// TIA Portal project "FactoryIO_Template_S7-1200_V16_V16" (V16)
// Vorlageprojekt für das Buch mit Zielsystem S7-1200

(* hardware
DEVICE "S7-1200-Station_1"  S7-1200 Station
   slot 0: "Baugruppenträger_0"  Rack  V1.0
   slot 1: "PLC_1"  CPU 1211C DC/DC/DC  6ES7 211-1AE40-0XB0  V4.1
*)

// ===== PLC "PLC_1"  CPU 1211C DC/DC/DC =====

VAR_GLOBAL   // PLC tag table "Standard-Variablentabelle"
   "Tag_4" AT %I10.0 : Bool;
   "Tag_5" AT %Q10.0 : Bool;
   "Tag_6" AT %I10.1 : Bool;
   "loop marker" AT %M0.0 : Bool;
   "stop-cond" AT %M0.1 : Bool;
   "stop-cond-pulse" AT %M0.2 : Bool;
   "Tag_1" AT %M2.0 : Bool;
   "Tag_2" AT %M2.1 : Bool;
   "cancel-grap" AT %M0.3 : Bool;
   "return-X" AT %M0.4 : Bool;
   "reset-c" AT %M0.5 : Bool;
   "Tag_7" AT %M2.2 : Bool;
   "Tag_8" AT %M1.0 : Bool;
   "Tag_9" AT %M1.1 : Bool;
   "grab-control" AT %M0.6 : Bool;
   "Tag_3" AT %M2.3 : Bool;
   "Tag_10" AT %M2.4 : Bool;
   "Tag_11" AT %M1.2 : Bool;
   "shift palett" AT %M0.7 : Bool;
   "Tag_12" AT %M2.5 : Bool;
   "palett-c-reset" AT %M1.3 : Bool;
   "Tag_13" AT %M2.6 : Bool;
END_VAR

VAR_GLOBAL   // PLC tag table "Tag table from XML_1"
   "Start Button" AT %I0.0 : Bool;
   "Stop Button" AT %I0.1 : Bool;
   "Emergency Stop" AT %I0.2 : Bool;
   "Diffuse Sensor 1" AT %I0.3 : Bool;
   "Diffuse Sensor 2" AT %I0.4 : Bool;
   "Diffuse Sensor 3" AT %I0.5 : Bool;
   "Moving (Z) Detected" AT %I0.6 : Bool;
   "Moving (X) Detected" AT %I0.7 : Bool;
   "Detected" AT %I1.0 : Bool;
   "Belt Conveyor 1 (6m)" AT %Q0.0 : Bool;
   "Belt Conveyor 2 (6m)" AT %Q0.1 : Bool;
   "Belt Conveyor (4m)" AT %Q0.2 : Bool;
   "Roller Conveyor 1 (6m)" AT %Q0.3 : Bool;
   "Roller Conveyor 2 (6m)" AT %Q0.4 : Bool;
   "Roller Conveyor (4m)" AT %Q0.5 : Bool;
   "Moving (Z)" AT %Q0.6 : Bool;
   "Moving (X)" AT %Q0.7 : Bool;
   "Grab" AT %Q1.0 : Bool;
   "Start Button  (Light)" AT %Q1.1 : Bool;
   "Stop Button  (Light)" AT %Q1.2 : Bool;
END_VAR

// folder: System blocks/Program resources

DATA_BLOCK "palett-c"   // DB1
{ S7_Optimized_Access := 'TRUE' }
AUTHOR : Simatic
FAMILY : IEC
NAME : CNTR
VERSION : 1.0
// stored: InstanceOfName IEC_COUNTER
"IEC_COUNTER"
BEGIN
END_DATA_BLOCK

DATA_BLOCK "sequence-counter"   // DB2
{ S7_Optimized_Access := 'TRUE' }
AUTHOR : Simatic
FAMILY : IEC
NAME : CNTR
VERSION : 1.0
// stored: InstanceOfName IEC_COUNTER
"IEC_COUNTER"
BEGIN
END_DATA_BLOCK

DATA_BLOCK "palett-shift"   // DB3
{ S7_Optimized_Access := 'TRUE' }
AUTHOR : Simatic
FAMILY : IEC
NAME : IEC_TMR
VERSION : 1.0
// stored: InstanceOfName IEC_TIMER
"IEC_TIMER"
BEGIN
END_DATA_BLOCK

DATA_BLOCK "TT"   // DB4
{ S7_Optimized_Access := 'TRUE' }
AUTHOR : Simatic
FAMILY : IEC
NAME : IEC_TMR
VERSION : 1.0
// stored: InstanceOfName IEC_TIMER
"IEC_TIMER"
BEGIN
END_DATA_BLOCK

// folder: (top level)

FUNCTION "MHJ-PLC-Lab-Function-S71200" : Void   // FC9000, SCL
{ S7_Optimized_Access := 'TRUE' }
VERSION : 0.1
   VAR_TEMP
      rdTimeReturn : Int;
      outputTime : DTL;
      SyncVal : Byte;
      forVal : Int;
      forVal_2 : Int;
      Value : Byte;
   END_VAR
   VAR CONSTANT
      CompVal : Byte := 16#34;
      Value_01 : Byte := 16#11;
      Value_01_DW : DWord := 16#A165_D992;
      Value_02_DW : DWord := 16#58BE_4401;
   END_VAR
BEGIN

   #Value:=PEEK(area := 16#82,
        dbNumber := 0,
        byteOffset := 511);
   #Value := #Value + 1;

   POKE(area := 16#82,
        dbNumber := 0,
        byteOffset := 511,
        value := #Value);

   POKE(area:=16#81,
        dbNumber:=0,
        byteOffset:=1016,
        value:=#Value_01_DW);
   POKE(area := 16#81,
        dbNumber := 0,
        byteOffset := 1020,
        value := #Value_02_DW);

   POKE(area := 16#81,
        dbNumber := 0,
        byteOffset := 511,
        value := B#16#00);

   FOR #forVal := 0 TO 120 DO
       FOR #forVal_2:=0 TO 10 DO
           #rdTimeReturn:=RD_SYS_T(#outputTime);
           #rdTimeReturn := WR_SYS_T(#outputTime);
           #rdTimeReturn := RD_SYS_T(#outputTime);
           #rdTimeReturn := WR_SYS_T(#outputTime);
       END_FOR;
       #SyncVal:= PEEK(area := 16#81,
                      dbNumber := 0,
                      byteOffset := 511);
       IF #SyncVal = #CompVal THEN
          GOTO M_1;
       END_IF;
   END_FOR;
   RETURN;

   M_1:
   POKE(area := 16#81,
        dbNumber := 0,
        byteOffset := 511,
        value := B#16#0);
END_FUNCTION

ORGANIZATION_BLOCK "Main"   // OB1, LAD, ProgramCycle
TITLE = "Main Program Sweep (Cycle)"
{ S7_Optimized_Access := 'TRUE' }
VERSION : 0.1
   VAR_INPUT
      Initial_Call : Bool;   // Initial call of this OB
      Remanence : Bool;   // =True, if remanent data are available
   END_VAR
   VAR_TEMP   // added for the SCL form of the ladder/FBD networks
      _w1 : Bool;
      _w2 : Bool;
   END_VAR
BEGIN

REGION Network 1: Konnektierungsbaustein für PLC-Lab
   // Im Netzwerk 1 wird der Konnektierungsbaustein für PLC-Lab aufgerufen.
   // Dieser Aufruf darf nicht entfernt werden!
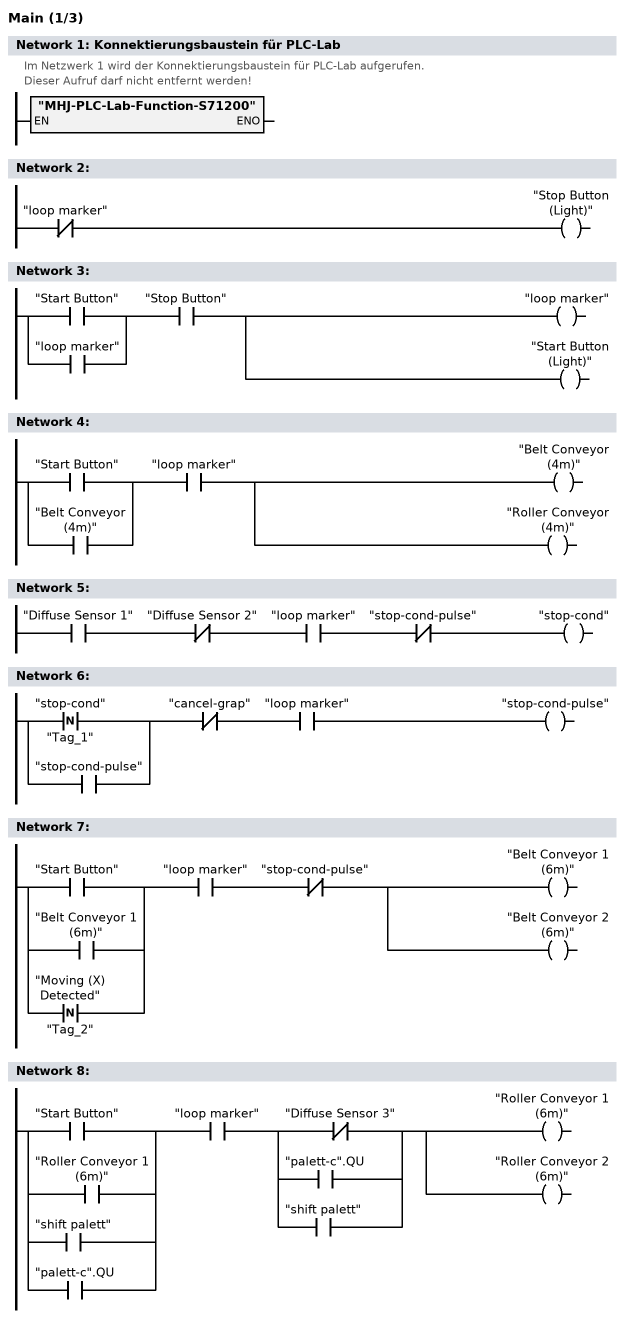
   RUNG wire#powerrail
      "MHJ-PLC-Lab-Function-S71200"()
   END_RUNG
   // the same network as SCL:
   "MHJ-PLC-Lab-Function-S71200"();
END_REGION

REGION Network 2
   RUNG wire#powerrail
      I_Contact( "loop marker" )
      Coil( "Stop Button  (Light)" )
   END_RUNG
   // the same network as SCL:
   "Stop Button  (Light)" := NOT "loop marker";
END_REGION

REGION Network 3
   RUNG wire#powerrail
      Contact( "Start Button" )
      wire#w1
      Contact( "Stop Button" )
      wire#w2
      Coil( "loop marker" )
   END_RUNG
   RUNG wire#powerrail
      Contact( "loop marker" )
   END_RUNG wire#w1
   RUNG wire#w2
      Coil( "Start Button  (Light)" )
   END_RUNG
   // the same network as SCL:
   "loop marker" := ("Start Button" OR "loop marker") AND "Stop Button";
   "Start Button  (Light)" := "loop marker";
END_REGION

REGION Network 4
   RUNG wire#powerrail
      Contact( "Start Button" )
      wire#w1
      Contact( "loop marker" )
      wire#w2
      Coil( "Belt Conveyor (4m)" )
   END_RUNG
   RUNG wire#powerrail
      Contact( "Belt Conveyor (4m)" )
   END_RUNG wire#w1
   RUNG wire#w2
      Coil( "Roller Conveyor (4m)" )
   END_RUNG
   // the same network as SCL:
   "Belt Conveyor (4m)" := ("Start Button" OR "Belt Conveyor (4m)") AND "loop marker";
   "Roller Conveyor (4m)" := "Belt Conveyor (4m)";
END_REGION

REGION Network 5
   RUNG wire#powerrail
      Contact( "Diffuse Sensor 1" )
      I_Contact( "Diffuse Sensor 2" )
      Contact( "loop marker" )
      I_Contact( "stop-cond-pulse" )
      Coil( "stop-cond" )
   END_RUNG
   // the same network as SCL:
   "stop-cond" := "Diffuse Sensor 1" AND NOT "Diffuse Sensor 2" AND "loop marker" AND NOT "stop-cond-pulse";
END_REGION

REGION Network 6
   RUNG wire#powerrail
      N_Contact(operand := "stop-cond", bit := "Tag_1")
      wire#w1
      I_Contact( "cancel-grap" )
      Contact( "loop marker" )
      Coil( "stop-cond-pulse" )
   END_RUNG
   RUNG wire#powerrail
      Contact( "stop-cond-pulse" )
   END_RUNG wire#w1
   // the same network as SCL:
   #_w1 := NOT "stop-cond" AND "Tag_1";   // falling edge of "stop-cond"
   "Tag_1" := "stop-cond";
   "stop-cond-pulse" := (#_w1 OR "stop-cond-pulse") AND NOT "cancel-grap" AND "loop marker";
END_REGION

REGION Network 7
   RUNG wire#powerrail
      Contact( "Start Button" )
      wire#w1
      Contact( "loop marker" )
      I_Contact( "stop-cond-pulse" )
      wire#w2
      Coil( "Belt Conveyor 1 (6m)" )
   END_RUNG
   RUNG wire#powerrail
      Contact( "Belt Conveyor 1 (6m)" )
   END_RUNG wire#w1
   RUNG wire#powerrail
      N_Contact(operand := "Moving (X) Detected", bit := "Tag_2")
   END_RUNG wire#w1
   RUNG wire#w2
      Coil( "Belt Conveyor 2 (6m)" )
   END_RUNG
   // the same network as SCL:
   #_w1 := NOT "Moving (X) Detected" AND "Tag_2";   // falling edge of "Moving (X) Detected"
   "Tag_2" := "Moving (X) Detected";
   "Belt Conveyor 1 (6m)" := ("Start Button" OR "Belt Conveyor 1 (6m)" OR #_w1) AND "loop marker" AND NOT "stop-cond-pulse";
   "Belt Conveyor 2 (6m)" := "Belt Conveyor 1 (6m)";
END_REGION

REGION Network 8
   RUNG wire#powerrail
      Contact( "Start Button" )
      wire#w1
      Contact( "loop marker" )
      wire#w2
      I_Contact( "Diffuse Sensor 3" )
      wire#w3
      Coil( "Roller Conveyor 1 (6m)" )
   END_RUNG
   RUNG wire#powerrail
      Contact( "Roller Conveyor 1 (6m)" )
   END_RUNG wire#w1
   RUNG wire#powerrail
      Contact( "shift palett" )
   END_RUNG wire#w1
   RUNG wire#powerrail
      Contact( "palett-c".QU )
   END_RUNG wire#w1
   RUNG wire#w2
      Contact( "palett-c".QU )
   END_RUNG wire#w3
   RUNG wire#w2
      Contact( "shift palett" )
   END_RUNG wire#w3
   RUNG wire#w3
      Coil( "Roller Conveyor 2 (6m)" )
   END_RUNG
   // the same network as SCL:
   "Roller Conveyor 1 (6m)" := ("Start Button" OR "Roller Conveyor 1 (6m)" OR "shift palett" OR "palett-c".QU) AND "loop marker" AND (NOT "Diffuse Sensor 3" OR "palett-c".QU OR "shift palett");
   "Roller Conveyor 2 (6m)" := "Roller Conveyor 1 (6m)";
END_REGION

REGION Network 9
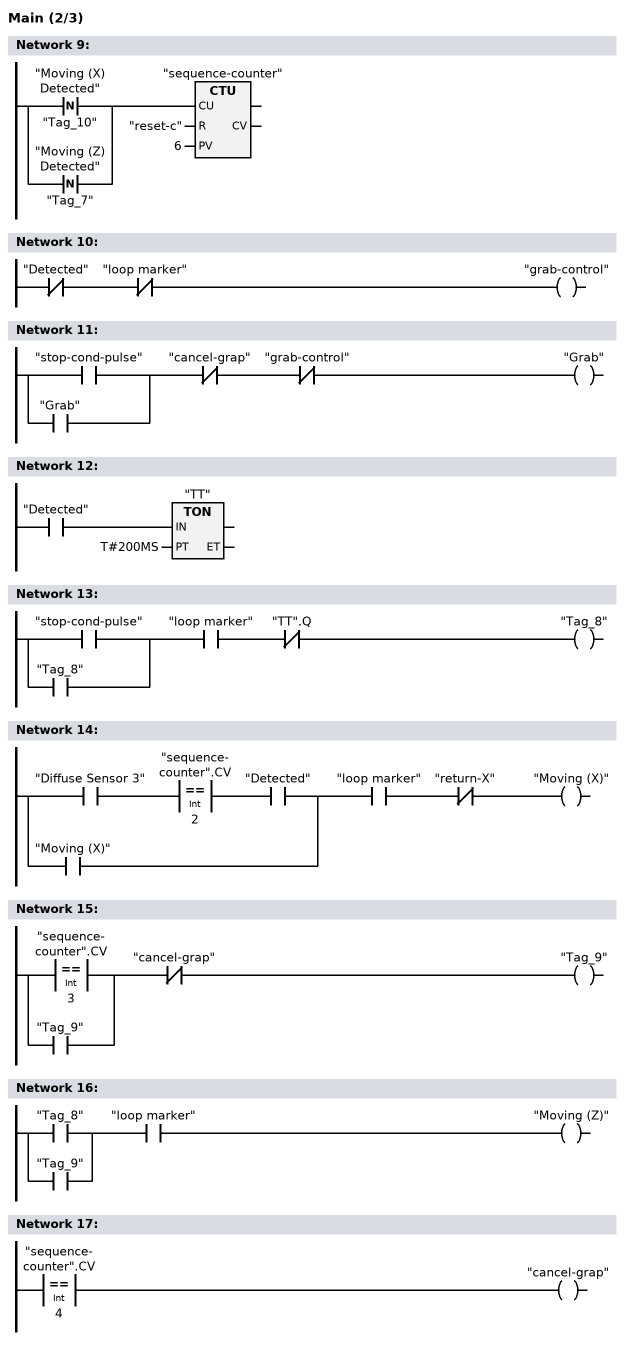
   #_w1 := NOT "Moving (X) Detected" AND "Tag_10";   // falling edge of "Moving (X) Detected"
   "Tag_10" := "Moving (X) Detected";
   #_w2 := NOT "Moving (Z) Detected" AND "Tag_7";   // falling edge of "Moving (Z) Detected"
   "Tag_7" := "Moving (Z) Detected";
   "sequence-counter".CTU(CU := #_w1 OR #_w2, R := "reset-c", PV := 6);
END_REGION

REGION Network 10
   RUNG wire#powerrail
      I_Contact( "Detected" )
      I_Contact( "loop marker" )
      Coil( "grab-control" )
   END_RUNG
   // the same network as SCL:
   "grab-control" := NOT "Detected" AND NOT "loop marker";
END_REGION

REGION Network 11
   RUNG wire#powerrail
      Contact( "stop-cond-pulse" )
      wire#w1
      I_Contact( "cancel-grap" )
      I_Contact( "grab-control" )
      Coil( "Grab" )
   END_RUNG
   RUNG wire#powerrail
      Contact( "Grab" )
   END_RUNG wire#w1
   // the same network as SCL:
   "Grab" := ("stop-cond-pulse" OR "Grab") AND NOT "cancel-grap" AND NOT "grab-control";
END_REGION

REGION Network 12
   "TT".TON(IN := "Detected", PT := T#200MS);
END_REGION

REGION Network 13
   RUNG wire#powerrail
      Contact( "stop-cond-pulse" )
      wire#w1
      Contact( "loop marker" )
      I_Contact( "TT".Q )
      Coil( "Tag_8" )
   END_RUNG
   RUNG wire#powerrail
      Contact( "Tag_8" )
   END_RUNG wire#w1
   // the same network as SCL:
   "Tag_8" := ("stop-cond-pulse" OR "Tag_8") AND "loop marker" AND NOT "TT".Q;
END_REGION

REGION Network 14
   RUNG wire#powerrail
      Contact( "Diffuse Sensor 3" )
      { S7_Templates := "SrcType := Int" } EQ_Contact(in1 := "sequence-counter".CV, in2 := 2)
      Contact( "Detected" )
      wire#w1
      Contact( "loop marker" )
      I_Contact( "return-X" )
      Coil( "Moving (X)" )
   END_RUNG
   RUNG wire#powerrail
      Contact( "Moving (X)" )
   END_RUNG wire#w1
   // the same network as SCL:
   "Moving (X)" := (("Diffuse Sensor 3" AND ("sequence-counter".CV = 2) AND "Detected") OR "Moving (X)") AND "loop marker" AND NOT "return-X";
END_REGION

REGION Network 15
   RUNG wire#powerrail
      { S7_Templates := "SrcType := Int" } EQ_Contact(in1 := "sequence-counter".CV, in2 := 3)
      wire#w1
      I_Contact( "cancel-grap" )
      Coil( "Tag_9" )
   END_RUNG
   RUNG wire#powerrail
      Contact( "Tag_9" )
   END_RUNG wire#w1
   // the same network as SCL:
   "Tag_9" := (("sequence-counter".CV = 3) OR "Tag_9") AND NOT "cancel-grap";
END_REGION

REGION Network 16
   RUNG wire#powerrail
      Contact( "Tag_8" )
      wire#w1
      Contact( "loop marker" )
      Coil( "Moving (Z)" )
   END_RUNG
   RUNG wire#powerrail
      Contact( "Tag_9" )
   END_RUNG wire#w1
   // the same network as SCL:
   "Moving (Z)" := ("Tag_8" OR "Tag_9") AND "loop marker";
END_REGION

REGION Network 17
   RUNG wire#powerrail
      { S7_Templates := "SrcType := Int" } EQ_Contact(in1 := "sequence-counter".CV, in2 := 4)
      Coil( "cancel-grap" )
   END_RUNG
   // the same network as SCL:
   "cancel-grap" := "sequence-counter".CV = 4;
END_REGION

REGION Network 18
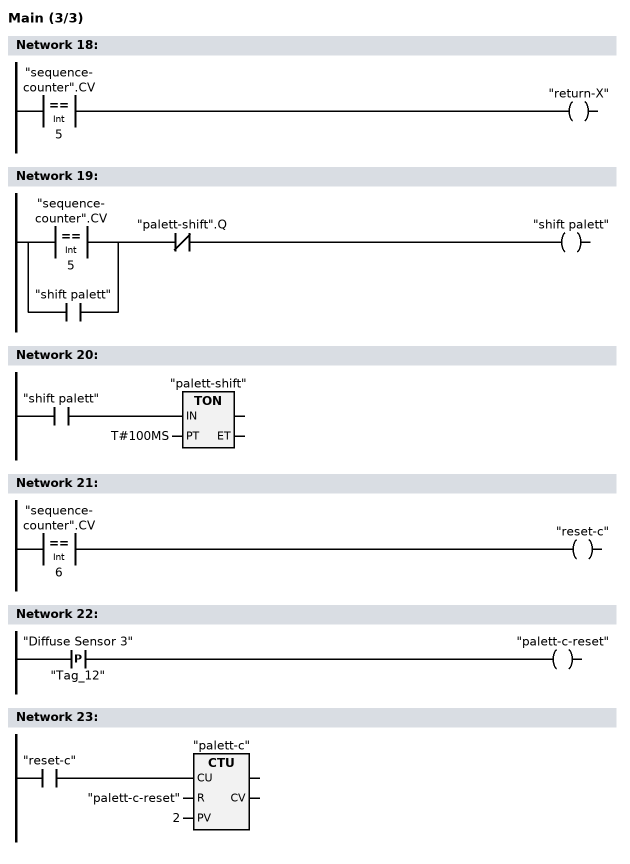
   RUNG wire#powerrail
      { S7_Templates := "SrcType := Int" } EQ_Contact(in1 := "sequence-counter".CV, in2 := 5)
      Coil( "return-X" )
   END_RUNG
   // the same network as SCL:
   "return-X" := "sequence-counter".CV = 5;
END_REGION

REGION Network 19
   RUNG wire#powerrail
      { S7_Templates := "SrcType := Int" } EQ_Contact(in1 := "sequence-counter".CV, in2 := 5)
      wire#w1
      I_Contact( "palett-shift".Q )
      Coil( "shift palett" )
   END_RUNG
   RUNG wire#powerrail
      Contact( "shift palett" )
   END_RUNG wire#w1
   // the same network as SCL:
   "shift palett" := (("sequence-counter".CV = 5) OR "shift palett") AND NOT "palett-shift".Q;
END_REGION

REGION Network 20
   "palett-shift".TON(IN := "shift palett", PT := T#100MS);
END_REGION

REGION Network 21
   RUNG wire#powerrail
      { S7_Templates := "SrcType := Int" } EQ_Contact(in1 := "sequence-counter".CV, in2 := 6)
      Coil( "reset-c" )
   END_RUNG
   // the same network as SCL:
   "reset-c" := "sequence-counter".CV = 6;
END_REGION

REGION Network 22
   RUNG wire#powerrail
      P_Contact(operand := "Diffuse Sensor 3", bit := "Tag_12")
      Coil( "palett-c-reset" )
   END_RUNG
   // the same network as SCL:
   #_w1 := "Diffuse Sensor 3" AND NOT "Tag_12";   // rising edge of "Diffuse Sensor 3"
   "Tag_12" := "Diffuse Sensor 3";
   "palett-c-reset" := #_w1;
END_REGION

REGION Network 23
   "palett-c".CTU(CU := "reset-c", R := "palett-c-reset", PV := 2);
END_REGION
END_ORGANIZATION_BLOCK